FUNCTION_BLOCK DigitalOutputParametersFB
VAR_INPUT
	DOut: DigitalOutputParameters;
END_VAR
VAR_OUTPUT
	H_GP1_OnTime: LTIME;
	F_QM1_OnTime: LTIME;
	F_QM2_OnTime: LTIME;
	T_QM2_OnTime: LTIME;
END_VAR
VAR
	H_GP1_LTON: Timer; // $(skip)
	F_QM1_LTON: Timer; // $(skip)
	F_QM2_LTON: Timer; // $(skip)
	T_QM2_LTON: Timer; // $(skip)
END_VAR

H_GP1_LTON(EN := DOut.H_GP1, ET => H_GP1_OnTime);
F_QM1_LTON(EN := DOut.F_QM1, ET => F_QM1_OnTime);
F_QM2_LTON(EN := DOut.F_QM2, ET => F_QM2_OnTime);
T_QM2_LTON(EN := DOut.T_QM2, ET => T_QM2_OnTime);

METHOD Update : BOOL
VAR_INPUT
	DO_: REFERENCE TO GreenMasterDO_Base;
	Parameters: REFERENCE TO GreenMasterBaseParameters;
	EnableWriteDampers: BOOL := TRUE;
END_VAR

DO_.H_GP1 := Parameters.IO.DOut.H_GP1;
DO_.C_GP1 := Parameters.IO.DOut.C_GP1;
IF EnableWriteDampers THEN
	DO_.F_QM1 := Parameters.IO.DOut.F_QM1;
	DO_.T_QM2 := Parameters.IO.DOut.T_QM2;
END_IF
DO_.R_QM1 := Parameters.IO.DOut.R_QM1;
DO_.F_QM2 := Parameters.IO.DOut.F_QM2;
DO_.T_QM1_1 := Parameters.IO.DOut.T_QM1_1;
DO_.T_QM1_2 := Parameters.IO.DOut.T_QM1_2;
DO_.T_QM1_3 := Parameters.IO.DOut.T_QM1_3;
DO_.T_QM1_4 := Parameters.IO.DOut.T_QM1_4;
DO_.T_QM1_5 := Parameters.IO.DOut.T_QM1_5;
DO_.T_QM1_6 := Parameters.IO.DOut.T_QM1_6;
Parameters.IO.DOut.F_QM2_ActiveWhenStopped := FALSE;
DO_.SupplyRunning := Parameters.IO.DOut.T_RUN;
DO_.ExhaustRunning := Parameters.IO.DOut.F_RUN;

DO_.AlarmRelayA := Parameters.IO.DOut.AL_A;
DO_.AlarmRelayB := Parameters.IO.DOut.AL_B;
DO_.AlarmRelayC := Parameters.IO.DOut.AL_C;
DO_.AlarmRelayD := Parameters.IO.DOut.AL_D;
END_METHOD

END_FUNCTION_BLOCK

(* stored: Version 1.1.0.1, ProductVersion 3.1.4024.6
   POU DigitalOutputParametersFB: Id {85648e1a-e841-444e-abc6-5abe348f319a}, SpecialFunc None
   Method Update: Id {c3e83810-423d-49ef-bca7-1df8d58ed7c0} *)
